
TYPE "DriveCalcSpeedOutput"
STRUCT
        calculatedSpeed : INT;
        isRunning : BOOL;
END_STRUCT;
END_TYPE